{attribute 'linkalways'} 
{attribute 'no_explicit_call' := 'This FB is a CLASS and must be accessed using methods or properties'}
{attribute 'enable_dynamic_creation'}
FUNCTION_BLOCK Node_F_VN_ApplyScalingToAffineTransformationExp EXTENDS VisionNode
VAR
    aTransformationMatrix : _TcVnMatrix2x3_LREAL;
    fScaleX : _LREAL(0.0);
    fScaleY : _LREAL(0.0);
    bUsePreMultiplication : _BOOL(FALSE);
    hrPrev : _HRESULT(S_OK);
	hresult : _HRESULT(S_OK);
END_VAR

METHOD PUBLIC  Clone : I_Node
VAR
	pNode : POINTER TO Node_F_VN_ApplyScalingToAffineTransformationExp;
END_VAR
pNode := __NEW(Node_F_VN_ApplyScalingToAffineTransformationExp);
Clone := pNode^;
END_METHOD

METHOD FB_init : BOOL
VAR_INPUT
	bInitRetains : BOOL; // if TRUE, the retain variables are initialized (warm start / cold start)
	bInCopyCode : BOOL;  // if TRUE, the instance afterwards gets moved into the copy code (online change)
END_VAR
AddInput('aTransformationMatrix', aTransformationMatrix);
AddParameter('fScaleX', fScaleX);
AddParameter('fScaleY', fScaleY);
AddParameter('bUsePreMultiplication', bUsePreMultiplication);
AddInput('hrPrev', hrPrev);
AddOutput('aTransformationMatrix', aTransformationMatrix);
AddOutput('hresult', hresult);
END_METHOD

METHOD PROTECTED  OnExecute : HRESULT
hresult.Value := F_VN_ApplyScalingToAffineTransformationExp(
	aTransformationMatrix := aTransformationMatrix.Value,
    fScaleX := fScaleX.Value,
    fScaleY := fScaleY.Value,
    bUsePreMultiplication := bUsePreMultiplication.Value,
	hrPrev := hrPrev.Value);
END_METHOD

METHOD PUBLIC PreExecutionCheck
VAR_INPUT
	Check : I_PreExecutionChecks;
END_VAR
END_METHOD

END_FUNCTION_BLOCK

(* stored: Version 1.1.0.1, ProductVersion 3.1.4024.13
   POU Node_F_VN_ApplyScalingToAffineTransformationExp: Id {c73c0c7c-a8dc-0d86-3e6b-c632e76714fa}, SpecialFunc None
   Folder Constructor: Id {f0aacdcf-4737-07c3-3e6a-402b4ef27c22}
   Method Clone: Id {cfb19155-ca93-0e17-081e-88cd9dd16c9c}
   Method FB_init: Id {13d41fbf-53ee-0864-1a67-d374860fbb88}
   Method OnExecute: Id {d9ec19e0-0c9b-04d7-341c-b699b7770693}
   Method PreExecutionCheck: Id {2f8e7feb-4d08-04e2-3888-9009db794abb} *)
